// TIA Portal project "Smart_Water_Tank_Project" (V16)

(* hardware
DEVICE "S71500/ET200MP-Station_1"  S7-1500 station
   slot 0: "Profilschiene_0"  Rack  6ES7 590-1***0-0AA0
   slot 1: "PLC_1"  CPU 1513-1 PN  6ES7 513-1AL02-0AB0  V2.8
      slot 3: "CPU-Display_1"  6ES7591-1AA00-0AA0
      slot 32768: "PROFINET-Schnittstelle_1"  X1
         slot 32769: "Port_1"  X1 P1
         slot 32770: "Port_2"  X1 P2
      slot 34817: "Virtual CP interface port_1"  Virtual CP interface port  Virtual CP interface port
   slot 2: "AI 8xU/I/RTD/TC ST_1"  AI 8xU/I/RTD/TC ST  6ES7 531-7KF00-0AB0  V2.0
   slot 3: "AI 8xU/I/RTD/TC ST_2"  AI 8xU/I/RTD/TC ST  6ES7 531-7KF00-0AB0  V2.0
   slot 4: "AI 8xU/I/RTD/TC ST_3"  AI 8xU/I/RTD/TC ST  6ES7 531-7KF00-0AB0  V2.0
   slot 5: "AI 8xU/I/RTD/TC ST_4"  AI 8xU/I/RTD/TC ST  6ES7 531-7KF00-0AB0  V2.0
   slot 6: "DI 16x24VDC BA_1"  DI 16x24VDC BA  6ES7 521-1BH10-0AA0  V1.0
*)

// ===== PLC "PLC_1"  CPU 1513-1 PN =====

VAR_GLOBAL   // PLC tag table "Standard-Variablentabelle"
   "Start" AT %I0.0 : Bool;
   "Motor" AT %Q0.0 : Bool;
   "Stop" AT %I0.1 : Bool;
   "Fill_Valve" AT %Q0.1 : Bool;
   "Fill_Green" AT %Q0.2 : Bool;
   "Discharge_PB" AT %I0.2 : Bool;
   "Dis_Valve" AT %Q0.3 : Bool;
   "Dis_Red" AT %Q0.4 : Bool;
   "Tag_1" AT %QW30 : Word;
   "Tag_2" AT %QD10 : DInt;
   "Fill_Valve_n" AT %QD100 : Real;
   "Tag_4" AT %M0.0 : Bool;
   "Tag_5" AT %M0.4 : Bool;
   "Level_Meter" AT %ID100 : Real;
   "Discharge_Valve" AT %QD104 : Real;
   "Tag_8" AT %QD34 : Real;
   "Tag_9" AT %QD30 : Real;
   "Tag_10" AT %ID30 : Real;
   "sys_Run" AT %M0.1 : Bool;
   "Statue" AT %MD0 : DInt;
END_VAR

DATA_BLOCK "DB_Tank"   // DB2
{ S7_Optimized_Access := 'TRUE' }
VERSION : 0.1
   VAR
      Tank_Level : Real := 0.0;
      Level_SP : Real := 0.0;
      Fill_Output : Real;
      Discharge_Output : Bool;
      Fill_Command : Real := 0.0;
      Fill_Rate : Real := 0.5;
      Discharge_Rate : Real := 0.5;
      PID_Mode : Int;
      Fill_Increment : Real;
      Auto_Mode : Bool;
      Manual_Start : Bool;
      Auto_Rising : Bool;
      Auto_Falling : Bool;
      PID_ModeActivate : Bool;
      Fill_Enable : Bool;
      Level_Raw : Real;
      Level_Error : Real;
      Discharge_Command : Real;
      Negative_Error : Real;
   END_VAR
BEGIN
END_DATA_BLOCK

FUNCTION "MHJ-PLC-Lab-Function-S71500" : Void   // FC9000, SCL
{ S7_Optimized_Access := 'TRUE' }
VERSION : 0.1
   VAR_TEMP
      Value : Byte;
      ForCounter : Int;
   END_VAR
   VAR CONSTANT
      Value_01_DW : DWord := 16#1223_5486;
      Value_02_DW : DWord := 16#A6C9_D1F5;
   END_VAR
BEGIN

   #Value:=PEEK(area := 16#82,
        dbNumber := 0,
        byteOffset := 511);
   #Value := #Value + 1;

   POKE(area := 16#82,
        dbNumber := 0,
        byteOffset := 511,
        value := #Value);

   POKE(area := 16#82,
        dbNumber := 0,
        byteOffset := 1016,
        value := #Value_01_DW);
   POKE(area := 16#82,
        dbNumber := 0,
        byteOffset := 1020,
        value := #Value_02_DW);

   FOR #ForCounter := 0 TO 63 DO
       #Value:=PEEK(area := 16#1,
            dbNumber := 0,
            byteOffset := #ForCounter);
       POKE(area := 16#81,
            dbNumber := 0,
            byteOffset := #ForCounter,
            value := #Value);
   END_FOR;
   #Value := PEEK(area := 16#1,
                  dbNumber := 0,
                  byteOffset := 512);
   POKE(area := 16#82,
        dbNumber := 0,
        byteOffset := 512,
        value := #Value);
END_FUNCTION

ORGANIZATION_BLOCK "Main"   // OB1, LAD, ProgramCycle
TITLE = "Main Program Sweep (Cycle)"
{ S7_Optimized_Access := 'TRUE' }
VERSION : 0.1
   VAR_INPUT
      Initial_Call : Bool;   // Initial call of this OB
      Remanence : Bool;   // =True, if remanent data are available
   END_VAR
BEGIN

REGION Network 1
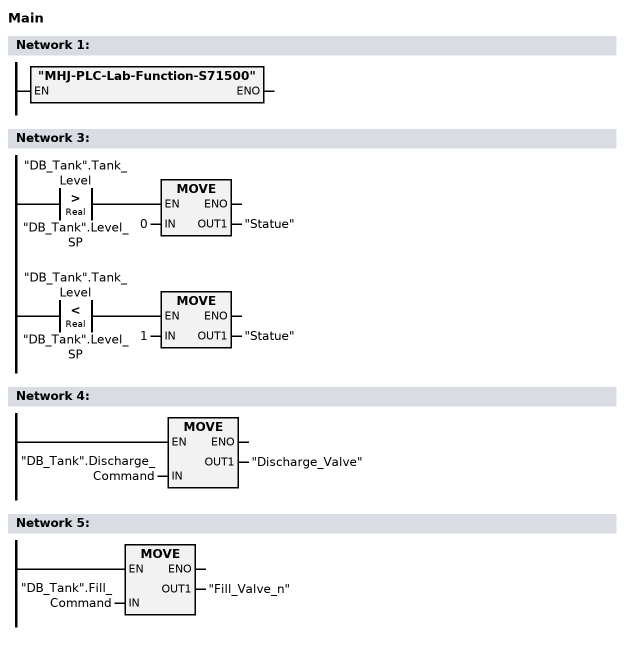
   RUNG wire#powerrail
      "MHJ-PLC-Lab-Function-S71500"()
   END_RUNG
   // the same network as SCL:
   "MHJ-PLC-Lab-Function-S71500"();
END_REGION

REGION Network 3
   RUNG wire#powerrail
      { S7_Templates := "SrcType := Real" } GT_Contact(in1 := "DB_Tank".Tank_Level, in2 := "DB_Tank".Level_SP)
      Move(in := 0, out1 => "Statue")
   END_RUNG
   RUNG wire#powerrail
      { S7_Templates := "SrcType := Real" } LT_Contact(in1 := "DB_Tank".Tank_Level, in2 := "DB_Tank".Level_SP)
      Move(in := 1, out1 => "Statue")
   END_RUNG
   // the same network as SCL:
   IF "DB_Tank".Tank_Level > "DB_Tank".Level_SP THEN "Statue" := 0; END_IF;
   IF "DB_Tank".Tank_Level < "DB_Tank".Level_SP THEN "Statue" := 1; END_IF;
END_REGION

REGION Network 4
   RUNG wire#powerrail
      Move(in := "DB_Tank".Discharge_Command, out1 => "Discharge_Valve")
   END_RUNG
   // the same network as SCL:
   "Discharge_Valve" := "DB_Tank".Discharge_Command;
END_REGION

REGION Network 5
   RUNG wire#powerrail
      Move(in := "DB_Tank".Fill_Command, out1 => "Fill_Valve_n")
   END_RUNG
   // the same network as SCL:
   "Fill_Valve_n" := "DB_Tank".Fill_Command;
END_REGION
END_ORGANIZATION_BLOCK

ORGANIZATION_BLOCK "Cyclic interrupt"   // OB30, LAD, CyclicInterrupt
{ S7_Optimized_Access := 'TRUE' }
VERSION : 0.1
   VAR_INPUT
      Initial_Call : Bool;   // Initial call of this OB
      Event_Count : Int;   // Events discarded
   END_VAR
BEGIN

REGION Network 1
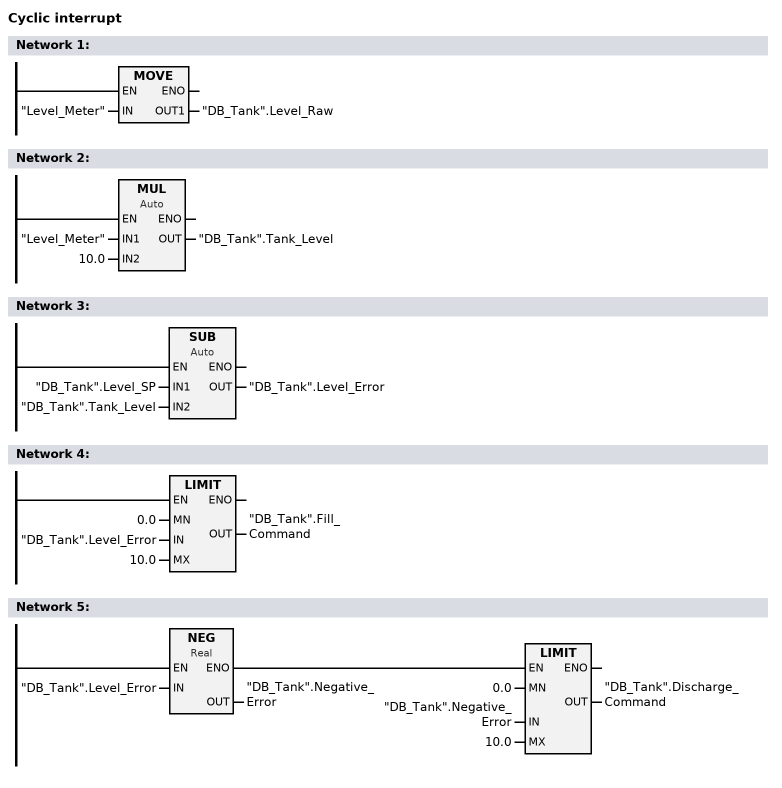
   RUNG wire#powerrail
      Move(in := "Level_Meter", out1 => "DB_Tank".Level_Raw)
   END_RUNG
   // the same network as SCL:
   "DB_Tank".Level_Raw := "Level_Meter";
END_REGION

REGION Network 2
   RUNG wire#powerrail
      Mul(in1 := "Level_Meter", in2 := 10.0, out => "DB_Tank".Tank_Level)
   END_RUNG
   // the same network as SCL:
   "DB_Tank".Tank_Level := "Level_Meter" * 10.0;
END_REGION

REGION Network 3
   RUNG wire#powerrail
      Sub(in1 := "DB_Tank".Level_SP, in2 := "DB_Tank".Tank_Level, out => "DB_Tank".Level_Error)
   END_RUNG
   // the same network as SCL:
   "DB_Tank".Level_Error := "DB_Tank".Level_SP - "DB_Tank".Tank_Level;
END_REGION

REGION Network 4
   "DB_Tank".Fill_Command := LIMIT(MN := 0.0, IN := "DB_Tank".Level_Error, MX := 10.0);
END_REGION

REGION Network 5
   "DB_Tank".Negative_Error := -"DB_Tank".Level_Error;
   "DB_Tank".Discharge_Command := LIMIT(MN := 0.0, IN := "DB_Tank".Negative_Error, MX := 10.0);
END_REGION
END_ORGANIZATION_BLOCK